FUNCTION_BLOCK PUBLIC Disposable_TestSuite EXTENDS TcUnit.FB_TestSuite
VAR
END_VAR

DisposedFromDisposeMethod();
DisposedByManuallyDeleting();

METHOD PUBLIC DisposedByManuallyDeleting
VAR
	mockDispose : POINTER TO MockDisposable;
	disposed : BOOL;
END_VAR
TEST('DisposedByManuallyDeleting');

// @TEST-FIXTURE
mockDispose := __NEW(MockDisposable(DisposedFlag:=disposed));

// @TEST-RUN
__DELETE(mockDispose);

// @TEST-ASSSERT
AssertTrue(
	Condition := disposed,
	Message := 'FB_exit was not correctly triggered in the MockDisposable'
);

TEST_FINISHED();
END_METHOD

METHOD PUBLIC DisposedFromDisposeMethod
VAR
	mockDispose : POINTER TO MockDisposable;
	disposed : BOOL;
END_VAR
TEST('DisposedFromDisposeMethod');

// @TEST-FIXTURE
mockDispose := __NEW(MockDisposable(DisposedFlag:=disposed));

// @TEST-RUN
mockDispose^.Dispose();

// @TEST-ASSSERT
AssertTrue(
	Condition := disposed,
	Message := 'FB_exit was not correctly triggered in the MockDisposable'
);

TEST_FINISHED();
END_METHOD

END_FUNCTION_BLOCK

(* stored: Version 1.1.0.1, ProductVersion 3.1.4024.12
   POU Disposable_TestSuite: Id {5e30d77d-5ab7-4a68-9932-9d53fc3729bd}, SpecialFunc None
   Method DisposedByManuallyDeleting: Id {53f28239-f13a-41de-aa9f-47d3ff4c2a4d}
   Method DisposedFromDisposeMethod: Id {f6d78085-e7eb-482f-b15d-638e7798de7e} *)
